// TIA Portal V18 export
DATA_BLOCK "AHUAlarms"   // DB101
{ S7_Optimized_Access := 'FALSE' }
VERSION : 0.1
// stored: AutoNumber false, DBAccessibleFromOPCUA true, IsOnlyStoredInLoadMemory false, IsWriteProtectedInAS false
   VAR
      Summary { S7_SetPoint := 'True'} : "UDT_AHUSummaryAlarms";
   END_VAR
BEGIN
END_DATA_BLOCK
